(*
	Handles communication and control of a Vaisala GMW90 environment sensor (Temp, Humidity, CO2)
*)
{attribute 'OPC.UA.DA.StructuredType' := '1'}
FUNCTION_BLOCK FB_Sensor_VaisalaGMW90_R2_1 EXTENDS FB_BaseDevice

VAR_INPUT
	nModbusUnitID: UINT; // slave ID of the sensor
END_VAR

VAR_IN_OUT
	fbModbusManager : FB_ModbusManager;
	
END_VAR

VAR_OUTPUT
	{attribute 'OPC.UA.DA' := '1'}
	rCO2 : REAL;
	{attribute 'OPC.UA.DA' := '1'}
	rTemperature : REAL;
	{attribute 'OPC.UA.DA' := '1'}
	rHumidity : REAL;

END_VAR

VAR PERSISTENT 
	tDataRefresh: TIME := T#1m;
	tWaitForReadings: TIME := T#17S;
	tWaitForTurnOff: TIME := T#100MS;
	tMsgTimeout: TIME := T#2S;
	bEnableComms: BOOL := FALSE;
END_VAR

VAR
	
	
	bReading: BOOL := FALSE;
	bFirstRun: BOOL := TRUE;
	bResetTtimer: BOOL := FALSE;
	
	nWordsToRead_values : UINT := 1; // ( CO2;  Temp;  Hum)
	nWordsToRead_errors : UINT := 2; // The GMW90 has 16 bits for error codes
	
	nAdrFirstReg_CO2 : WORD := 256; // THE GMW90 stores its int value for CO2 value in register 256
	nAdrFirstReg_Hum : WORD := 257; // THE GMW90 stores its int value for CO2 value in register 256
	nAdrFirstReg_Temp : WORD := 258; // THE GMW90 stores its int value for CO2 value in register 256
	
	nAdrFirstReg_Error : WORD := 513; // the GMW90 stores its error codes in 0513 register
	
	stModRequest_ReadCO2: ST_Modbus_ReadRequest;
	stModRequest_ReadHum: ST_Modbus_ReadRequest;
	stModRequest_ReadTemp: ST_Modbus_ReadRequest;
	
	stModRequest_ReadError: ST_Modbus_ReadRequest;
	
	bVaisalaPowerCtr AT %Q*: BOOL;
	
	
	eSMState: (WAIT, ON, READ, TURN_OFF) := WAIT;
	
	fbTON_WaitForReadings: TON := (PT := tWaitForReadings, IN := FALSE);
	fbTON_WaitForTurnOff: TON := (PT := tWaitForReadings, IN := FALSE);
	fbTON_DataRefresh: TON := (PT := tDataRefresh, IN := FALSE);
	fbTON_MsgTimeout: TON := (PT := tMsgTimeout, IN := FALSE);
END_VAR

fbTON_WaitForTurnOff(PT := tWaitForTurnOff);
fbTON_WaitForReadings(PT := tWaitForReadings);
fbTON_DataRefresh(PT := tDataRefresh);
fbTON_MsgTimeout(PT := tMsgTimeout);

bVaisalaPowerCtr := TRUE;		// THis is a remnant of the power cycle workaround implemented in R7, keep this line here until we rewire room 7

IF bEnableComms THEN 
	IF bFirstRun THEN
		fbTON_DataRefresh(IN := TRUE);
		bFirstRun := FALSE;
		init_ModbusRequests();
	END_IF
	
	IF bResetTtimer THEN
		fbTON_DataRefresh(IN := TRUE);
		bResetTtimer := FALSE;
	END_IF
	
	(*
	IF nModbusUnitID <> 0 THEN
		bEnableComms := TRUE;
	END_IF
	*)
	
	CASE eSMState OF
		WAIT:
			fbTON_DataRefresh(IN := TRUE, PT := tDataRefresh);
			IF fbTON_DataRefresh.Q THEN
				eSMState := ON;
				fbTON_DataRefresh(IN := FALSE);
			END_IF
		
		ON:
			fbTON_WaitForReadings(PT := tWaitForReadings, IN := TRUE);
			//bVaisalaPowerCtr := TRUE;
			IF fbTON_WaitForReadings.Q THEN
				eSMState := READ;
			END_IF
			
		READ:
			IF fbTON_WaitForReadings.Q THEN
				fbTON_WaitForReadings(IN := FALSE);
				fbModbusManager.addRequest_Read_Vaisala(ReadRequest := ADR(stModRequest_ReadCO2));
				fbTON_MsgTimeout(IN := TRUE);
			END_IF
			
			IF stModRequest_ReadCO2.bRequestCompleted OR fbTON_MsgTimeout.Q THEN
				stModRequest_ReadCO2.bRequestCompleted := FALSE;
				fbTON_MsgTimeout( IN := FALSE);
				fbTON_WaitForTurnOff(IN := TRUE);
			END_IF
			
			IF fbTON_WaitForTurnOff.Q THEN
				//bVaisalaPowerCtr := FALSE;
				eSMState := WAIT;
				fbTON_WaitForTurnOff(IN := FALSE);
			END_IF
			
	END_CASE
	
	rCO2 := 			stModRequest_ReadCO2.ReadRegsVals[1]; 
	rHumidity :=  		stModRequest_ReadCO2.ReadRegsVals[2] / 100.00; 
	rTemperature := 	stModRequest_ReadCO2.ReadRegsVals[3] / 100.00; 
	
	
	(*
	
	IF fbTON_DataRefresh.Q AND bEnableComms THEN
		
		IF NOT fbTON_WaitForReadings.Q AND NOT bReading THEN
			fbTON_WaitForReadings(IN := TRUE);
			bVaisalaPowerCtr := TRUE;				// Turn the vaisala unit on
			bReading := TRUE;
		END_IF
			
		IF fbTON_WaitForReadings.Q THEN			// We have waited for the unit to power on, now we read
			fbModbusManager.addRequest_Read_Vaisala(ReadRequest := ADR(stModRequest_ReadCO2));
			fbTON_WaitForReadings(IN := FALSE);
		END_IF
		
		IF (stModRequest_ReadCO2.bRequestCompleted = TRUE) THEN // Request has finished, we turn power off after a set amount of time
			stModRequest_ReadCO2.bRequestCompleted := FALSE;
			fbTON_WaitForTurnOff(IN := TRUE);
		END_IF
		IF fbTON_WaitForTurnOff.Q THEN
			bVaisalaPowerCtr := FALSE;
			fbTON_WaitForTurnOff(IN := FALSE);
			fbTON_DataRefresh(IN := FALSE); 
			bResetTtimer := TRUE;
			fbTON_WaitForReadings(IN := FALSE);
			bReading := FALSE;
		END_IF
	END_IF
		
		
	
		//fbModbusManager.addRequest_Read(ReadRequest := ADR(stModRequest_ReadError));
		
		//fbModbusManager.addRequest_Read_Vaisala(ReadRequest := ADR(stModRequest_ReadCO2));
		//fbModbusManager.addRequest_Read_Vaisala(ReadRequest := ADR(stModRequest_ReadCO2));
		
		
	*)
END_IF

METHOD init_ModbusRequests : BOOL
VAR_INPUT
END_VAR
stModRequest_ReadCO2.SlaveAddress := nModbusUnitID;			
stModRequest_ReadCO2.AdrFirstSlaveRegisterRead := nAdrFirstReg_CO2;
stModRequest_ReadCO2.QtyWordsToRead := 3;				
stModRequest_ReadCO2.bRequestAccepted := FALSE;
stModRequest_ReadCO2.bRequestCompleted := FALSE;
stModRequest_ReadCO2.ReadRegsVals := GVL.ModbusEmptyBuffer;

(*
stModRequest_ReadHum.SlaveAddress := nModbusUnitID;			
stModRequest_ReadHum.AdrFirstSlaveRegisterRead := nAdrFirstReg_Hum;
stModRequest_ReadHum.QtyWordsToRead := 1;				
stModRequest_ReadHum.bRequestAccepted := FALSE;
stModRequest_ReadHum.bRequestCompleted := FALSE;
stModRequest_ReadHum.ReadRegsVals := GVL.ModbusEmptyBuffer;

stModRequest_ReadTemp.SlaveAddress := nModbusUnitID;			
stModRequest_ReadTemp.AdrFirstSlaveRegisterRead := nAdrFirstReg_Temp;
stModRequest_ReadTemp.QtyWordsToRead := 1;				
stModRequest_ReadTemp.bRequestAccepted := FALSE;
stModRequest_ReadTemp.bRequestCompleted := FALSE;
stModRequest_ReadTemp.ReadRegsVals := GVL.ModbusEmptyBuffer;
*)

stModRequest_ReadError.SlaveAddress := nModbusUnitID;			
stModRequest_ReadError.AdrFirstSlaveRegisterRead := nAdrFirstReg_Error;
stModRequest_ReadError.QtyWordsToRead := nWordsToRead_errors;			
stModRequest_ReadError.bRequestAccepted := FALSE;
stModRequest_ReadError.bRequestCompleted := FALSE;
stModRequest_ReadError.ReadRegsVals := GVL.ModbusEmptyBuffer;
END_METHOD

END_FUNCTION_BLOCK

(* stored: Version 1.1.0.1, ProductVersion 3.1.4024.12
   POU FB_Sensor_VaisalaGMW90_R2_1: Id {db10d21e-45b8-43e0-aed4-cec00049eaab}, SpecialFunc None
   Method init_ModbusRequests: Id {4f636ca9-3f60-4569-9083-7d1c97afdea1} *)
